# EPICS substitutions: tdkLambda/slowDevicesApp/Db/template.substitutions
# template.substitutions
# Template file for Tdk Lambda
# Mehmet Bozdogan 04/11/2017
#
# substitutions:
# sys    - system
# sec    - section
# dev    - device
# $(sys)-$(sec)-$(dev) - device port(devPort)
#
#
################################################################################
file db/tdklambda.template {
    pattern 	{ sys	sec	dev	drvhV	drvlV	drvhC	drvlC	}
        	{ SYS	SEC	DEV	20	0	10	0	}
}
